// TIA Portal V15.1 export
// export: Created 2024-06-21T08:41:05.7351409Z, ExportSetting WithDefaults, DisplayName Totally Integrated Automation Portal, DisplayVersion V15.1 Update 5, DisplayName TIA Portal Openness, DisplayVersion V15.1 Update 5, DisplayName SINAMICS Startdrive Advanced, DisplayVersion V15.1, DisplayName G130, G150, S120, S150, SINAMICS MV, S210, DisplayVersion V15.1, DisplayName G110M, G120, G120C, G120D, G120P, DisplayVersion V15.1, DisplayName STEP 7 Professional, DisplayVersion V15.1 Update 5, DisplayName STEP 7 Safety, DisplayVersion V15.1, DisplayName WinCC Professional, DisplayVersion V15.1 Update 5, DisplayName SIMATIC Visualization Architect, DisplayVersion V15.1
FUNCTION_BLOCK "LGBSEW-MDXPN-6PD"   // FB6637, FBD
TITLE = LGBSEW-MDXPN-6PD
{ S7_Optimized_Access := 'TRUE' }
VERSION : 0.1
// =============================================================================
// This Module Handles LGBSEW-MDXPNSynch With DFS21B/DFS22B
// =============================================================================
// stored: AutoNumber false, IsIECCheckEnabled false, IsRetainMemResEnabled false, MemoryReserve 100, SetENOAutomatically False, UDAEnableTagReadback false
   VAR_INPUT
      I_OFF2 { ExternalAccessible := 'False'; ExternalVisible := 'False'; ExternalWritable := 'False'} : Bool;   // Rapid stop
      I_JogPositive { ExternalAccessible := 'False'; ExternalVisible := 'False'; ExternalWritable := 'False'} : Bool;   // Jog +
      I_JogNegative { ExternalAccessible := 'False'; ExternalVisible := 'False'; ExternalWritable := 'False'} : Bool;   // Jog -
      I_SynchMode { ExternalAccessible := 'False'; ExternalVisible := 'False'; ExternalWritable := 'False'} : Bool;   // Synchronisation Mode
      I_ResetFault { ExternalAccessible := 'False'; ExternalVisible := 'False'; ExternalWritable := 'False'} : Bool;   // Reset fault
      I_SetPointSpeed { ExternalAccessible := 'False'; ExternalVisible := 'False'; ExternalWritable := 'False'} : Int;   // Setpoint Speed mm/s
      I_Ramp { ExternalAccessible := 'False'; ExternalVisible := 'False'; ExternalWritable := 'False'} : Time;   // Ramp send in miliseconds (range : 100-10000ms, if 0 then default 1s will be used)
   END_VAR
   VAR_OUTPUT
      O_DriveReady { ExternalAccessible := 'False'; ExternalVisible := 'False'; ExternalWritable := 'False'} : Bool;   // Ready
      O_Active { ExternalAccessible := 'False'; ExternalVisible := 'False'; ExternalWritable := 'False'} : Bool;   // Active
      O_Alarm { ExternalAccessible := 'False'; ExternalVisible := 'False'; ExternalWritable := 'False'} : Bool;   // Alarm
      O_Warning { ExternalAccessible := 'False'; ExternalVisible := 'False'; ExternalWritable := 'False'} : Bool;   // Warning
      O_AlarmABCondition { ExternalAccessible := 'False'; ExternalVisible := 'False'; ExternalWritable := 'False'} : Bool;   // Alarm AB Condition
      O_AxisInterlocked { ExternalAccessible := 'False'; ExternalVisible := 'False'; ExternalWritable := 'False'} : Bool;   // Interlocked
      H_StatusWord { ExternalAccessible := 'False'; ExternalVisible := 'False'; ExternalWritable := 'False'} : Word;   // Status word from drive
      H_ControlWord { ExternalAccessible := 'False'; ExternalVisible := 'False'; ExternalWritable := 'False'} : Word;   // Control word to drive
      H_SetPointSpeed { ExternalAccessible := 'False'; ExternalVisible := 'False'; ExternalWritable := 'False'} : Int;   // Speed setpoint for drive
      H_SetpointSpeedProCent { ExternalAccessible := 'False'; ExternalVisible := 'False'; ExternalWritable := 'False'} : Real;   // Speed setpoint for drive %
      H_SetpointRamp { ExternalAccessible := 'False'; ExternalVisible := 'False'; ExternalWritable := 'False'} : Int;   // Ramp setpoint for drive
      H_ActualSpeed { ExternalAccessible := 'False'; ExternalVisible := 'False'; ExternalWritable := 'False'} : Real;   // Actual speed
      H_ActualCurrentA { ExternalAccessible := 'False'; ExternalVisible := 'False'; ExternalWritable := 'False'} : Real;   // Actual current Ampere
      H_ActualCurrentProCent { ExternalAccessible := 'False'; ExternalVisible := 'False'; ExternalWritable := 'False'} : Real;   // Actual current %
      H_ActualWarning { ExternalAccessible := 'False'; ExternalVisible := 'False'; ExternalWritable := 'False'} : Int;   // Actual Warning From Drive
      H_ActualFault { ExternalAccessible := 'False'; ExternalVisible := 'False'; ExternalWritable := 'False'} : Int;   // Actual Fault From Drive
   END_VAR
   VAR_IN_OUT
      C_HWSubInput { ExternalAccessible := 'False'; ExternalVisible := 'False'; ExternalWritable := 'False'} : HW_SUBMODULE;   // Config
      C_HWSubOutput { ExternalAccessible := 'False'; ExternalVisible := 'False'; ExternalWritable := 'False'} : HW_SUBMODULE;   // Config
      C_DriveCurrent { ExternalAccessible := 'False'; ExternalVisible := 'False'; ExternalWritable := 'False'} : Real;   // Reference current of the drive
      C_MotorCurrent { ExternalAccessible := 'False'; ExternalVisible := 'False'; ExternalWritable := 'False'} : Real;   // Reference current of the motor
   END_VAR
   VAR
      InputTelegram { ExternalAccessible := 'False'; ExternalVisible := 'False'; ExternalWritable := 'False'} : Struct   // Inputs telegram 6PD
         PI1 { ExternalAccessible := 'False'; ExternalVisible := 'False'; ExternalWritable := 'False'} : Struct   // Status word
            Status { ExternalAccessible := 'False'; ExternalVisible := 'False'; ExternalWritable := 'False'} : Byte;   // Status / error code
            DriveSynchronised { ExternalAccessible := 'False'; ExternalVisible := 'False'; ExternalWritable := 'False'} : Bool;   // Drive is synchronised
            InverterReady { ExternalAccessible := 'False'; ExternalVisible := 'False'; ExternalWritable := 'False'} : Bool;   // Inverter power section is ready for operation
            IPOSReferenced { ExternalAccessible := 'False'; ExternalVisible := 'False'; ExternalWritable := 'False'} : Bool;   // IPOS Referenced
            TargetPositionReached { ExternalAccessible := 'False'; ExternalVisible := 'False'; ExternalWritable := 'False'} : Bool;   // Target Position Reached
            BrakeReleased { ExternalAccessible := 'False'; ExternalVisible := 'False'; ExternalWritable := 'False'} : Bool;   // Brake Released
            FaultWarning { ExternalAccessible := 'False'; ExternalVisible := 'False'; ExternalWritable := 'False'} : Bool;   // Fault/warning present
            LimitSwitchCW { ExternalAccessible := 'False'; ExternalVisible := 'False'; ExternalWritable := 'False'} : Bool;   // Limit Switch CW
            LimitSwitchCCW { ExternalAccessible := 'False'; ExternalVisible := 'False'; ExternalWritable := 'False'} : Bool;   // Limit Switch CCW
         END_STRUCT;
         ActualPosition { ExternalAccessible := 'False'; ExternalVisible := 'False'; ExternalWritable := 'False'} : DInt;   // Actual Position
         ActualSpeed { ExternalAccessible := 'False'; ExternalVisible := 'False'; ExternalWritable := 'False'} : Int;   // Actual Speed
         PositionError { ExternalAccessible := 'False'; ExternalVisible := 'False'; ExternalWritable := 'False'} : Int;   // Position Error
         OutputCurrent { ExternalAccessible := 'False'; ExternalVisible := 'False'; ExternalWritable := 'False'} : Int;   // Output Current
      END_STRUCT;
      OutputTelegram { ExternalAccessible := 'False'; ExternalVisible := 'False'; ExternalWritable := 'False'} : Struct   // Outputs telegram 6PD
         PO1 { ExternalAccessible := 'False'; ExternalVisible := 'False'; ExternalWritable := 'False'} : Struct   // Control word
            Start { ExternalAccessible := 'False'; ExternalVisible := 'False'; ExternalWritable := 'False'} : Bool;   // Start
            JogPlus { ExternalAccessible := 'False'; ExternalVisible := 'False'; ExternalWritable := 'False'} : Bool;   // Jog +
            JogMinus { ExternalAccessible := 'False'; ExternalVisible := 'False'; ExternalWritable := 'False'} : Bool;   // Jog -
            Mode0 { ExternalAccessible := 'False'; ExternalVisible := 'False'; ExternalWritable := 'False'} : Bool;   // Mode
            Mode1 { ExternalAccessible := 'False'; ExternalVisible := 'False'; ExternalWritable := 'False'} : Bool;   // Mode
            CTW_Bit13 { ExternalAccessible := 'False'; ExternalVisible := 'False'; ExternalWritable := 'False'} : Bool;   // Reserved / not used
            CTW_Bit14 { ExternalAccessible := 'False'; ExternalVisible := 'False'; ExternalWritable := 'False'} : Bool;   // Reserved / not used
            CTW_Bit15 { ExternalAccessible := 'False'; ExternalVisible := 'False'; ExternalWritable := 'False'} : Bool;   // Reserved / not used
            ContrInhibit { ExternalAccessible := 'False'; ExternalVisible := 'False'; ExternalWritable := 'False'} : Bool;   // Interlock to drive
            RapidStop { ExternalAccessible := 'False'; ExternalVisible := 'False'; ExternalWritable := 'False'} : Bool;   // Rapid stop with stop ramp t13/t23, brake applied after stop
            Stop { ExternalAccessible := 'False'; ExternalVisible := 'False'; ExternalWritable := 'False'} : Bool;   // Stop to drive at normal ramp
            CTW_Bit3 { ExternalAccessible := 'False'; ExternalVisible := 'False'; ExternalWritable := 'False'} : Bool;   // Reserved / not used
            CTW_Bit4 { ExternalAccessible := 'False'; ExternalVisible := 'False'; ExternalWritable := 'False'} : Bool;   // Reserved / not used
            CTW_Bit5 { ExternalAccessible := 'False'; ExternalVisible := 'False'; ExternalWritable := 'False'} : Bool;   // Reserved / not used
            ResetFault { ExternalAccessible := 'False'; ExternalVisible := 'False'; ExternalWritable := 'False'} : Bool;   // Reset fault on drive
            CTW_Bit7 { ExternalAccessible := 'False'; ExternalVisible := 'False'; ExternalWritable := 'False'} : Bool;   // Reserved / not used
         END_STRUCT;
         TargetPosition { ExternalAccessible := 'False'; ExternalVisible := 'False'; ExternalWritable := 'False'} : DInt;   // Target position
         SetpointSpeed { ExternalAccessible := 'False'; ExternalVisible := 'False'; ExternalWritable := 'False'} : Int;   // Speed setpoint for drive (-4000-0-4000hex)
         Ramp { ExternalAccessible := 'False'; ExternalVisible := 'False'; ExternalWritable := 'False'} : Int;   // Ramp setpoint for drive
         Offset { ExternalAccessible := 'False'; ExternalVisible := 'False'; ExternalWritable := 'False'} : Int;   // Offset
      END_STRUCT;
      DriveWarning { ExternalAccessible := 'False'; ExternalVisible := 'False'; ExternalWritable := 'False'} : Bool;   // Drive Warning
      DriveAlarm { ExternalAccessible := 'False'; ExternalVisible := 'False'; ExternalWritable := 'False'} : Bool;   // Drive Alarm
      SynchMode { ExternalAccessible := 'False'; ExternalVisible := 'False'; ExternalWritable := 'False'} : Bool;   // Synchronisation Mode
      InverterCond { ExternalAccessible := 'False'; ExternalVisible := 'False'; ExternalWritable := 'False'} : Bool;   // Alarm AB Condition
      _Inverter { ExternalAccessible := 'False'; ExternalVisible := 'False'; ExternalWritable := 'False'} : "L1AlarmMultiIn";   // FB
   END_VAR
   VAR_TEMP
      TempReal : Real;   // Temp Real
      H_HMITemp : "H_HMI";   // Temp
   END_VAR
   VAR_TEMP   // added for the SCL form of the ladder/FBD networks
      _w1 : Bool;
   END_VAR
BEGIN

REGION Network 1: **** 1 - Inputs **** Read I/O Data
   // Read I/O Data
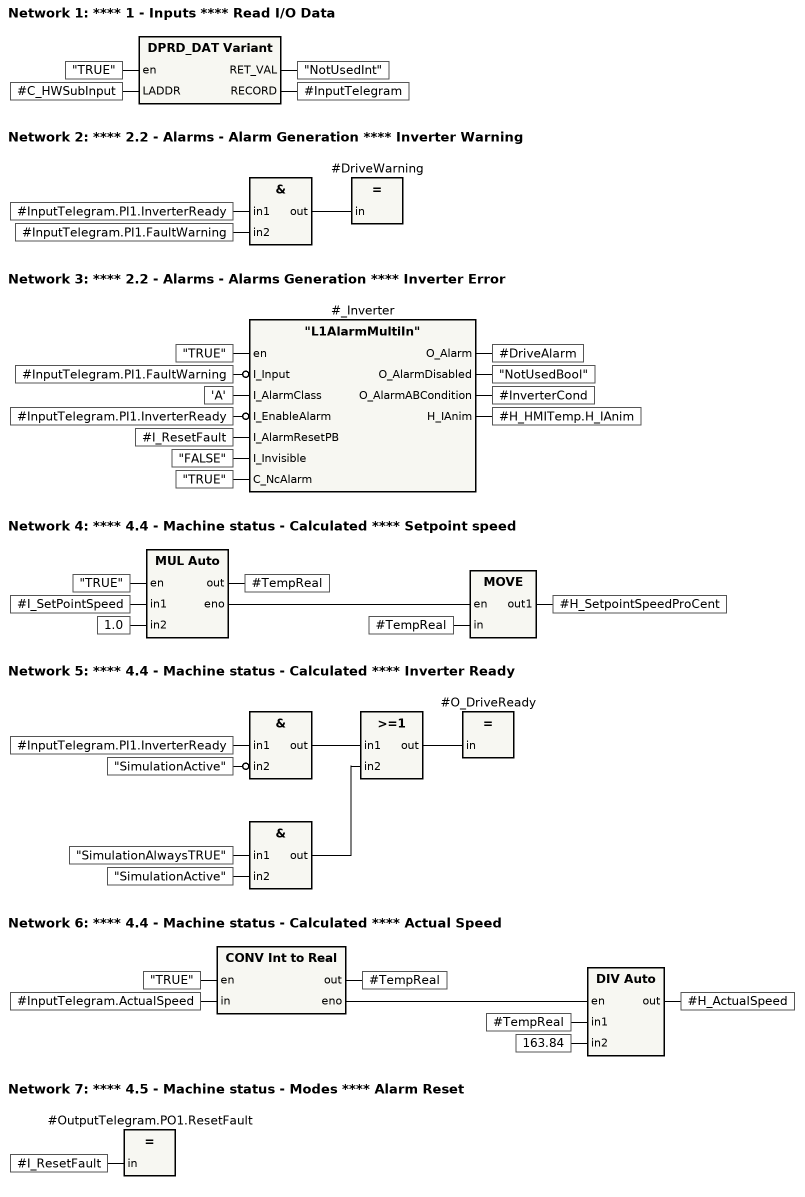
   IF "TRUE" THEN "NotUsedInt" := DPRD_DAT(LADDR := #C_HWSubInput, RECORD => #InputTelegram); END_IF;
END_REGION

REGION Network 2: **** 2.2 - Alarms - Alarm Generation **** Inverter Warning
   // Inverter  Warning
   #DriveWarning := #InputTelegram.PI1.InverterReady AND #InputTelegram.PI1.FaultWarning;
END_REGION

REGION Network 3: **** 2.2 - Alarms - Alarms Generation **** Inverter Error
   // Inverter Error
   IF "TRUE" THEN
       #_Inverter(I_Input := NOT #InputTelegram.PI1.FaultWarning,   // "L1AlarmMultiIn"
                  I_AlarmClass := 'A',
                  I_EnableAlarm := NOT #InputTelegram.PI1.InverterReady,
                  I_AlarmResetPB := #I_ResetFault,
                  I_Invisible := "FALSE",
                  C_NcAlarm := "TRUE",
                  O_Alarm => #DriveAlarm,
                  O_AlarmDisabled => "NotUsedBool",
                  O_AlarmABCondition => #InverterCond,
                  H_IAnim => #H_HMITemp.H_IAnim);
   END_IF;
END_REGION

REGION Network 4: **** 4.4 - Machine status - Calculated **** Setpoint speed
   // Convert Data
   IF "TRUE" THEN
       #TempReal := #I_SetPointSpeed * 1.0;
       #H_SetpointSpeedProCent := #TempReal;
   END_IF;
END_REGION

REGION Network 5: **** 4.4 - Machine status - Calculated **** Inverter Ready
   // Inverter Ready
   #O_DriveReady := (#InputTelegram.PI1.InverterReady AND NOT "SimulationActive") OR ("SimulationAlwaysTRUE" AND "SimulationActive");
END_REGION

REGION Network 6: **** 4.4 - Machine status - Calculated **** Actual Speed
   // Actual Speed
   IF "TRUE" THEN
       #TempReal := INT_TO_REAL(#InputTelegram.ActualSpeed);
       #H_ActualSpeed := #TempReal / 163.84;
   END_IF;
END_REGION

REGION Network 7: **** 4.5 - Machine status - Modes **** Alarm Reset
   // Alarm Reset
   #OutputTelegram.PO1.ResetFault := #I_ResetFault;
END_REGION

REGION Network 8: **** 4.6 - Machine status - Indication **** Status Word
   // Status Word
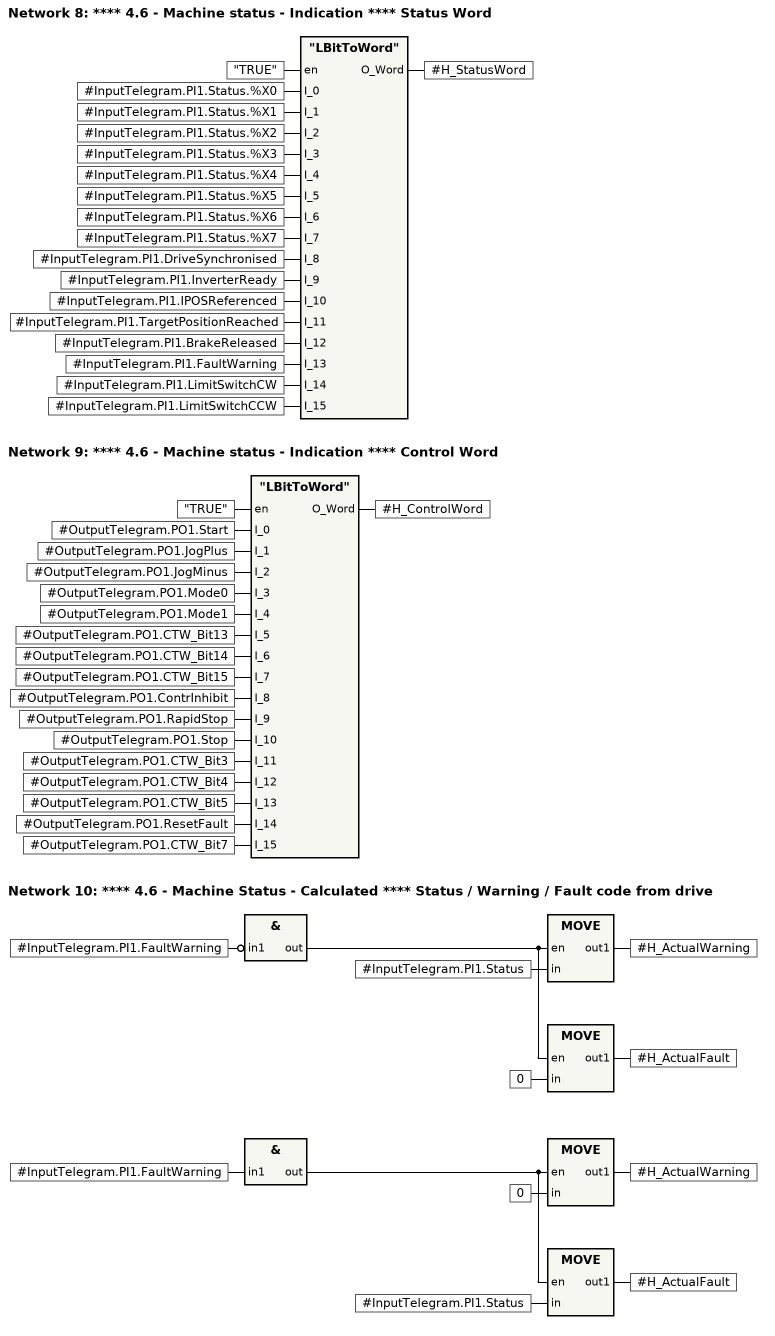
   IF "TRUE" THEN
       "LBitToWord"(I_0 := #InputTelegram.PI1.Status.%X0,
                    I_1 := #InputTelegram.PI1.Status.%X1,
                    I_2 := #InputTelegram.PI1.Status.%X2,
                    I_3 := #InputTelegram.PI1.Status.%X3,
                    I_4 := #InputTelegram.PI1.Status.%X4,
                    I_5 := #InputTelegram.PI1.Status.%X5,
                    I_6 := #InputTelegram.PI1.Status.%X6,
                    I_7 := #InputTelegram.PI1.Status.%X7,
                    I_8 := #InputTelegram.PI1.DriveSynchronised,
                    I_9 := #InputTelegram.PI1.InverterReady,
                    I_10 := #InputTelegram.PI1.IPOSReferenced,
                    I_11 := #InputTelegram.PI1.TargetPositionReached,
                    I_12 := #InputTelegram.PI1.BrakeReleased,
                    I_13 := #InputTelegram.PI1.FaultWarning,
                    I_14 := #InputTelegram.PI1.LimitSwitchCW,
                    I_15 := #InputTelegram.PI1.LimitSwitchCCW,
                    O_Word => #H_StatusWord);
   END_IF;
END_REGION

REGION Network 9: **** 4.6 - Machine status - Indication **** Control Word
   // Control Word
   IF "TRUE" THEN
       "LBitToWord"(I_0 := #OutputTelegram.PO1.Start,
                    I_1 := #OutputTelegram.PO1.JogPlus,
                    I_2 := #OutputTelegram.PO1.JogMinus,
                    I_3 := #OutputTelegram.PO1.Mode0,
                    I_4 := #OutputTelegram.PO1.Mode1,
                    I_5 := #OutputTelegram.PO1.CTW_Bit13,
                    I_6 := #OutputTelegram.PO1.CTW_Bit14,
                    I_7 := #OutputTelegram.PO1.CTW_Bit15,
                    I_8 := #OutputTelegram.PO1.ContrInhibit,
                    I_9 := #OutputTelegram.PO1.RapidStop,
                    I_10 := #OutputTelegram.PO1.Stop,
                    I_11 := #OutputTelegram.PO1.CTW_Bit3,
                    I_12 := #OutputTelegram.PO1.CTW_Bit4,
                    I_13 := #OutputTelegram.PO1.CTW_Bit5,
                    I_14 := #OutputTelegram.PO1.ResetFault,
                    I_15 := #OutputTelegram.PO1.CTW_Bit7,
                    O_Word => #H_ControlWord);
   END_IF;
END_REGION

REGION Network 10: **** 4.6 - Machine Status - Calculated **** Status / Warning / Fault code from drive
   // When the fault input is "True"   then the status code send over the byte is a fault code as decimal.
   // When the fault input is "False" then the status code send over the byte is a warning / status code as decimal.
   IF NOT #InputTelegram.PI1.FaultWarning THEN
       #H_ActualWarning := #InputTelegram.PI1.Status;
       #H_ActualFault := 0;
   END_IF;
   IF #InputTelegram.PI1.FaultWarning THEN
       #H_ActualWarning := 0;
       #H_ActualFault := #InputTelegram.PI1.Status;
   END_IF;
END_REGION

REGION Network 11: **** 5.1 - Equations - Interlock **** Interlock Axis
   // Interlock Axis
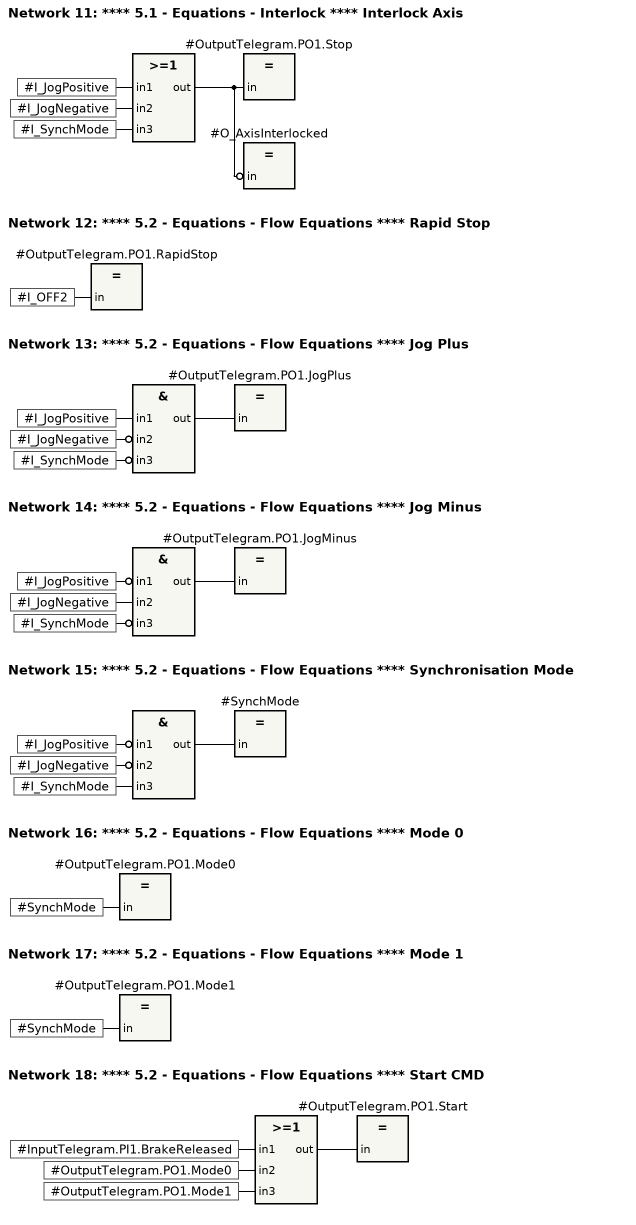
   #OutputTelegram.PO1.Stop := #I_JogPositive OR #I_JogNegative OR #I_SynchMode;
   #O_AxisInterlocked := NOT #OutputTelegram.PO1.Stop;
END_REGION

REGION Network 12: **** 5.2 - Equations - Flow Equations **** Rapid Stop
   // Rapid Stop
   #OutputTelegram.PO1.RapidStop := #I_OFF2;
END_REGION

REGION Network 13: **** 5.2 - Equations - Flow Equations **** Jog Plus
   // Jog Plus
   #OutputTelegram.PO1.JogPlus := #I_JogPositive AND NOT #I_JogNegative AND NOT #I_SynchMode;
END_REGION

REGION Network 14: **** 5.2 - Equations - Flow Equations **** Jog Minus
   // Jog Minus
   #OutputTelegram.PO1.JogMinus := NOT #I_JogPositive AND #I_JogNegative AND NOT #I_SynchMode;
END_REGION

REGION Network 15: **** 5.2 - Equations - Flow Equations **** Synchronisation Mode
   // Positioning Mode
   #SynchMode := NOT #I_JogPositive AND NOT #I_JogNegative AND #I_SynchMode;
END_REGION

REGION Network 16: **** 5.2 - Equations - Flow Equations **** Mode 0
   // Mode 0
   #OutputTelegram.PO1.Mode0 := #SynchMode;
END_REGION

REGION Network 17: **** 5.2 - Equations - Flow Equations **** Mode 1
   // Mode 1
   #OutputTelegram.PO1.Mode1 := #SynchMode;
END_REGION

REGION Network 18: **** 5.2 - Equations - Flow Equations **** Start CMD
   // Start CMD
   #OutputTelegram.PO1.Start := #InputTelegram.PI1.BrakeReleased OR #OutputTelegram.PO1.Mode0 OR #OutputTelegram.PO1.Mode1;
END_REGION

REGION Network 19: **** 5.2 - Equations - Flow Equations **** Reset All Commands Not Used
   // Reset All Commands Not Used
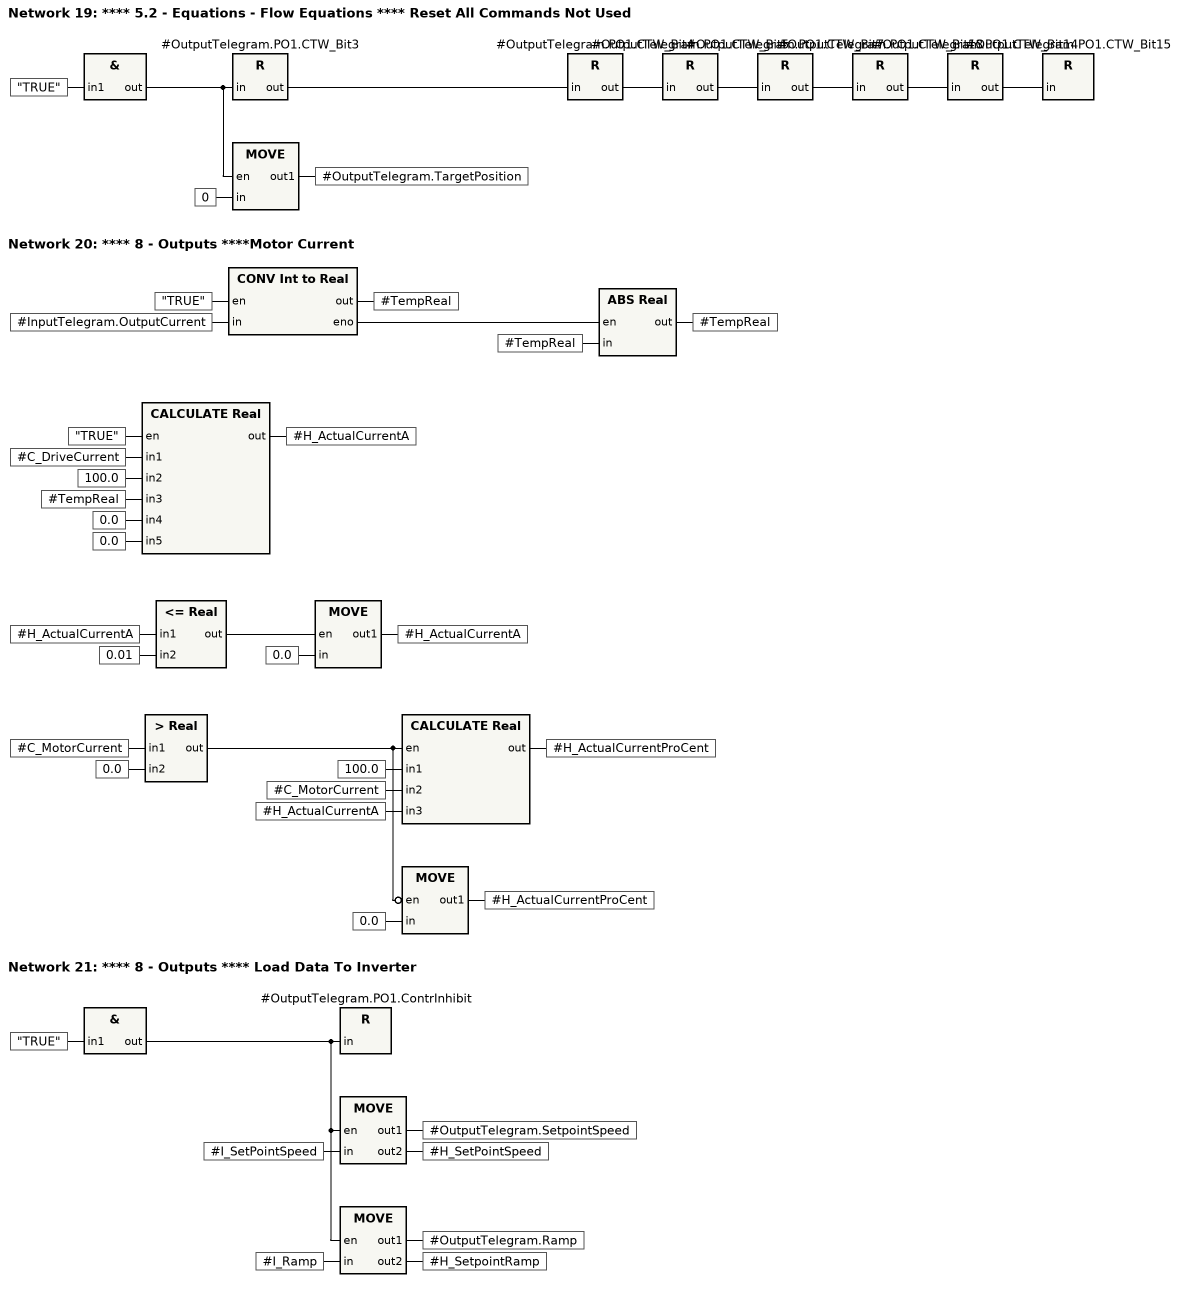
   IF "TRUE" THEN
       #OutputTelegram.PO1.CTW_Bit3 := FALSE;
       #OutputTelegram.PO1.CTW_Bit4 := FALSE;
       #OutputTelegram.PO1.CTW_Bit5 := FALSE;
       #OutputTelegram.PO1.CTW_Bit7 := FALSE;
       #OutputTelegram.PO1.CTW_Bit13 := FALSE;
       #OutputTelegram.PO1.CTW_Bit14 := FALSE;
       #OutputTelegram.PO1.CTW_Bit15 := FALSE;
       #OutputTelegram.TargetPosition := 0;
   END_IF;
END_REGION

REGION Network 20: **** 8 - Outputs ****Motor Current
   // Motor Current in % compared to the drive reference current (not the motor reference current)
   IF "TRUE" THEN
       #TempReal := INT_TO_REAL(#InputTelegram.OutputCurrent);
       #TempReal := ABS(#TempReal);   // Motor Current in % compared to the drive reference current (not the motor reference current) Remove - sign and use absolute value. Then scale this to the correct value (divide by 10 to get %) (This needs to be done since the drive can only send intiger values and not real values, so the drive does the percentage x10 to give a value behind the comma.) Then scale the % to a Ampere value and a % value compared to the motor reference current.
       #H_ActualCurrentA := #C_DriveCurrent - (((100.0 - #TempReal) / (100.0 - 0.0)) * (#C_DriveCurrent- 0.0));
   END_IF;
   IF #H_ActualCurrentA <= 0.01 THEN #H_ActualCurrentA := 0.0; END_IF;
   #_w1 := #C_MotorCurrent > 0.0;
   IF #_w1 THEN #H_ActualCurrentProCent := (100.0 / #C_MotorCurrent) * #H_ActualCurrentA; END_IF;
   IF NOT #_w1 THEN #H_ActualCurrentProCent := 0.0; END_IF;
END_REGION

REGION Network 21: **** 8 - Outputs **** Load Data To Inverter
   // Load Data To Inverter
   IF "TRUE" THEN
       #OutputTelegram.PO1.ContrInhibit := FALSE;
       #OutputTelegram.SetpointSpeed := #I_SetPointSpeed;
       #H_SetPointSpeed := #I_SetPointSpeed;
       #OutputTelegram.Ramp := #I_Ramp;
       #H_SetpointRamp := #I_Ramp;
   END_IF;
END_REGION

REGION Network 22: **** 8 - Outputs **** Alarm AB Condition
   // Alarm AB condition
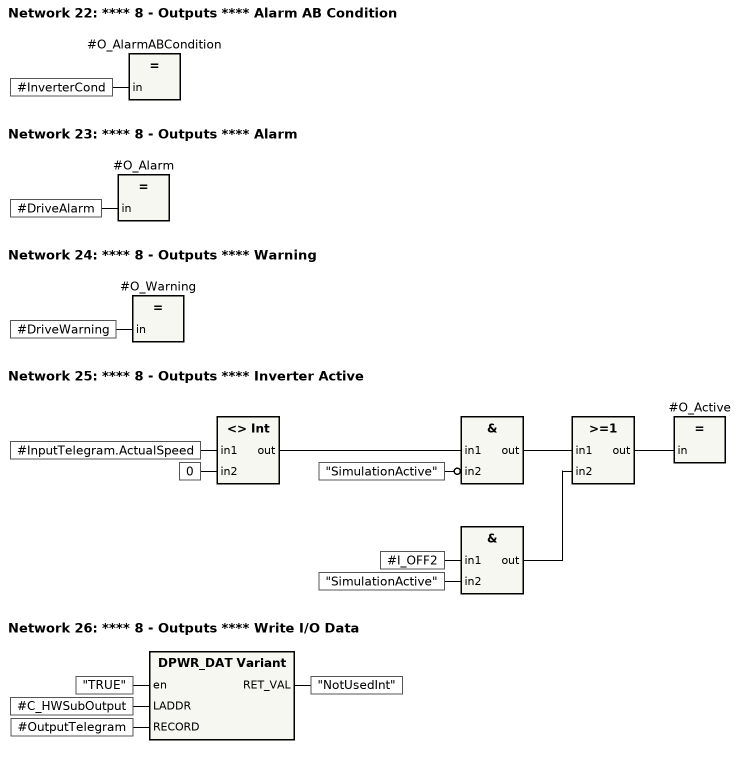
   #O_AlarmABCondition := #InverterCond;
END_REGION

REGION Network 23: **** 8 - Outputs **** Alarm
   // Alarm
   #O_Alarm := #DriveAlarm;
END_REGION

REGION Network 24: **** 8 - Outputs **** Warning
   // Warning
   #O_Warning := #DriveWarning;
END_REGION

REGION Network 25: **** 8 - Outputs **** Inverter Active
   // Inverter Active
   #O_Active := ((#InputTelegram.ActualSpeed <> 0) AND NOT "SimulationActive") OR (#I_OFF2 AND "SimulationActive");
END_REGION

REGION Network 26: **** 8 - Outputs **** Write I/O Data
   // Write I/O Data
   IF "TRUE" THEN "NotUsedInt" := DPWR_DAT(LADDR := #C_HWSubOutput, RECORD := #OutputTelegram); END_IF;
END_REGION
END_FUNCTION_BLOCK
